// TIA Portal V20 export
TYPE "typeSequenceControlNode_jrOutPnPRight"
// stored: Namespace Unit1.Em2
   STRUCT
      jobs : "LAF_typeJobs";
      sequence : "LAF_typeSequence";
      selectJobStatus { S7_SetPoint := 'True'} : Array[0..10] of "LAF_typeJobStatus";
      "step" : "LER_typeStep";
      jobInterface : "Unit1.Em2.typeSequenceControlNodeJobInterface_jrOutPnPRight";
      homeCheck : "Unit1.Em2.typeSequenceControlNodeHomeCheck_jrOutPnPRight";
   END_STRUCT;
   // // "step".action1[101] : Step[101] : JOB[1] Condition
   // // "step".action1[110] : Step[110] : JR PP Right Clamp Open
   // // "step".action1[130] : Step[130] : JR PP Right Clamp Close
   // // "step".action1[170] : Step[170] : JR PP Right Z-Axis Wait Pos
   // // "step".action1[180] : Step[180] : JR PP Right X-Axis Wait Pos
   // // "step".action1[190] : Step[190] : JOB[1] Step End
   // // "step".action1[201] : Step[201] : JOB[2] Condition
   // // "step".action1[210] : Step[210] : JR PP Right X-Axis Loading Pos[Top Tape Fix Stage]
   // // "step".action1[211] : Step[211] : JR PP Right Z-Axis Loading Pos[Top Tape Fix Stage]
   // // "step".action1[220] : Step[220] : JR PP Right [Loading Ready] => Top Tape Fix Stage
   // // "step".action1[221] : Step[221] : JR PP Right Clamp Close
   // // "step".action1[280] : Step[280] : JR PP Right X/Z-Axis Wait Pos
   // // "step".action1[290] : Step[290] : JOB[2] Step End
   // // "step".action1[301] : Step[301] : JOB[3] Condition
   // // "step".action1[310] : Step[310] : JR PP Right X-Axis Put Pos
   // // "step".action1[311] : Step[311] : JR PP Right Z-Axis Put Pos
   // // "step".action1[320] : Step[320] : JR PP Right [Unloading Ready] => Side Tape Fix Stage
   // // "step".action1[321] : Step[321] : JR PP Right Clamp Open
   // // "step".action1[322] : Step[322] : JR PP Right [Unclamp Done] => Side Tape Fix Stage
   // // "step".action1[380] : Step[380] : JR PP Right X/Z-Axis Wait Pos
   // // "step".action1[390] : Step[390] : JOB[3] Step End
   // // "step".transition1[101] : Step[101] : JOB[1] Condition
   // // "step".transition1[110] : Step[110] : JR PP Right Clamp Open
   // // "step".transition1[130] : Step[130] : JR PP Right Clamp Close
   // // "step".transition1[170] : Step[170] : JR PP Right Z-Axis Wait Pos
   // // "step".transition1[180] : Step[180] : JR PP Right X-Axis Wait Pos
   // // "step".transition1[190] : Step[190] : JOB[1] Step End
   // // "step".transition1[201] : Step[201] : JOB[2] Condition
   // // "step".transition1[210] : Step[210] : JR PP Right X-Axis Loading Pos[Top Tape Fix Stage]
   // // "step".transition1[211] : Step[211] : JR PP Right Z-Axis Loading Pos[Top Tape Fix Stage]
   // // "step".transition1[220] : Step[220] : JR PP Right [Loading Ready] => Top Tape Fix Stage
   // // "step".transition1[221] : Step[221] : JR PP Right Clamp Close
   // // "step".transition1[222] : Step[222] : JR PP Right [Clamp Done] => Top Tape Fix Stage
   // // "step".transition1[280] : Step[280] : JR PP Right X/Z-Axis Wait Pos
   // // "step".transition1[290] : Step[290] : JOB[2] Step End
   // // "step".transition1[301] : Step[301] : JOB[3] Condition
   // // "step".transition1[310] : Step[310] : JR PP Right X-Axis Put Pos
   // // "step".transition1[311] : Step[311] : JR PP Right Z-Axis Put Pos
   // // "step".transition1[320] : Step[320] : JR PP Right [Unloading Ready] => Side Tape Fix Stage
   // // "step".transition1[321] : Step[321] : JR PP Right Clamp Open
   // // "step".transition1[322] : Step[322] : JR PP Right [Unclamp Done] => Side Tape Fix Stage
   // // "step".transition1[380] : Step[380] : JR PP Right X/Z-Axis Wait Pos
   // // "step".transition1[390] : Step[390] : JOB[3] Step End
END_TYPE
